{attribute addProperty BoxType "EL1702-0000-0016"}
{attribute addProperty Id "ChannelAT %I*ARRAY[0..1] OF Channel_E4AEF59E1620WcStateAT %I*WcState_F855686C1620InfoDataAT %I*InfoData_192954DE1620"}
{attribute addProperty CRC "426425702"}
{attribute addProperty SizeInBites "48"}
{attribute addProperty SizeInBytes "6"}
TYPE EL1702_FE5AE676 :
STRUCT
	{attribute addProperty Name "Channel"}
	Channel : ARRAY[0..1] OF Channel_E4AEF59E;
	{attribute addProperty Name "WcState"}
	WcState : WcState_F855686C;
	{attribute addProperty Name "InfoData"}
	InfoData : InfoData_192954DE;
END_STRUCT
END_TYPE

(* stored: Version 1.2.0.0, ProductVersion 3.1.4024.9
   DUT EL1702_FE5AE676: Id {21fa3e55-10f5-44d3-895b-cd8d3e6b0da6} *)
